TYPE ST_PullOutConveyorInfo :
STRUCT
	ConveyorRunningTime : TIME; // This variable is the operating time of the conveyor belt forward.
	ConveyorReverseTime : TIME; // This variable is the operating time of the conveyor belt reverse.
	CommandType : E_PullOutConveyorCommandType; // Select PullOut conveyor command.
END_STRUCT
END_TYPE

(* stored: Version 1.1.0.1, ProductVersion 3.1.4024.13
   DUT ST_PullOutConveyorInfo: Id {3b9a0d9a-b042-4ee3-8e3f-373494209aad} *)
